TYPE IShortTest : 
STRUCT
	bStart :BOOL; //
	bDone  :BOOL; //

   iResult:INT; // 1 OK  2 NG
    
   ErrorID :INT;
   
	

END_STRUCT
END_TYPE

(* stored: Version 1.1.0.1, ProductVersion 3.1.4024.9
   DUT IShortTest: Id {463b0f28-7f5f-4ef2-93aa-01e736297f65} *)
